# B&R Automation Studio project AsClientTest
Automation Studio 4.9

## Configuration Config1

CPU X20CP0484, AutomationRuntime H4.93, Build 4.1.2, Vc V4.72.6

### Task classes (Cpu.sw)
```
Cyclic#1 (cycle 5000 us, tolerance 10000000 us):
  uaCltTest <- uaCltTest.prg
Libraries: EasyUaClnt, AsIecCon, runtime, astime, AsOpcUac, standard, AsBrStr
```

### Hardware
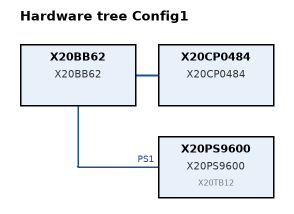
```
X20BB62 : X20BB62 v1.3.0.0
X20CP0484 : X20CP0484 v1.7.0.0  [SL -> X20BB62.SL1]
  Connector IF2:
    ActivateDevice = 1
    Mode = Manual
    InternetAddress = 192.168.2.10
    SubnetMask = 255.255.255.0
    ActivateSnmp = 2
  ConfigurationID = opcuaMethodCall_Config1
  Simulation = 1
  TimerDeviceType = SWIOTIMER
  TaskClassIdleTime = 10000
  CyclicTaskClassCount = 2
  Cyclic1Duration = 5000
  Cyclic1Tolerance = 10000000
  Cyclic2Duration = 20000
  Cyclic2Tolerance = 20000
  Cyclic3Duration = 50000
  Cyclic3Tolerance = 50000
  Cyclic4Duration = 100000
  Cyclic4Tolerance = 100000
  Cyclic5Duration = 200000
  Cyclic5Tolerance = 200000
  Cyclic6Duration = 500000
  Cyclic6Tolerance = 500000
  Cyclic7Duration = 1000000
  Cyclic7Tolerance = 1000000
  Cyclic8Duration = 10000
  Cyclic8Tolerance = 30000000
  FileDevice1
  FileDeviceName1 = USER
  FileDevicePath1 = USER_PATH
  ActivateOpcUa = 1
  OpcUaInformationModels_PV_Version = 1
X20PS9600 : X20PS9600 v1.6.1.0  [PS -> X20BB62.PS1; SS1 -> X20TB12.SS]
X20TB12 : X20TB12 v1.0.0.0
```

## Logical view

Binary libraries used (declarations not repeated): operator, runtime, astime, AsIecCon, EasyUaClnt 1.02.0, AsOpcUac, standard, AsBrStr


### Program Logical/uaCltTest (IEC)

#### Types.typ
```iecst
TYPE
	Sweep_typ : 	STRUCT
		input : Sweep_input_typ;
		output : Sweep_output_typ;
	END_STRUCT;
	Sweep_input_typ : 	STRUCT
		StartFrequency : LREAL;
		StopFrequency : LREAL;
		SweepPoints : DINT;
		SourceLevel : LREAL;
	END_STRUCT;
	Sweep_output_typ : 	STRUCT
		QFactor : LREAL;
		ResonanceFrequency : LREAL;
		Bandwidth : LREAL;
	END_STRUCT;
END_TYPE
```

#### Variables.var
```iecst
VAR CONSTANT
	MAX_OPCUA_CLIENTS : USINT := 9;
END_VAR
VAR
	EasyUaReads : ARRAY[0..MAX_OPCUA_CLIENTS] OF EasyUaRead;
	TON_0 : TON;
	Test : BOOL;
	i : USINT;
END_VAR
(*Variables to read into*)
VAR
	myBool : BOOL;
	myUsint : USINT;
	mySint : SINT;
	myUint : UINT;
	myInt : INT;
	myDint : DINT;
	myUdint : UDINT;
	myReal : REAL;
	myString : STRING[80];
END_VAR
```

#### Main.st
```iecst
// CLIENT SAMPLE TASK to read out the nodes from a OPCUA server.

PROGRAM _INIT
	// Setup for all clients
	FOR i:=0 TO MAX_OPCUA_CLIENTS DO
		EasyUaReads[i].ServerEndpointUrl := 'opc.tcp://127.0.0.2:4840'; // Don't use 127.0.0.1 as AS simulator put the server here as default.
		EasyUaReads[i].NamespaceUri := 'http://brdk.opcua.com';			// Specified on the server.
		EasyUaReads[i].NodeID.IdentifierType := UAIdentifierType_String;
	END_FOR

	// Setup for each node
	myBool;
	EasyUaReads[0].NodeID.Identifier := 'myBool';
	EasyUaReads[0].Variable := '::uaCltTest:myBool';

	myUsint;
	EasyUaReads[1].NodeID.Identifier := 'myUsint';
	EasyUaReads[1].Variable := '::uaCltTest:myUsint';

	mySint;
	EasyUaReads[2].NodeID.Identifier := 'mySint';
	EasyUaReads[2].Variable := '::uaCltTest:mySint';

	myUint;
	EasyUaReads[3].NodeID.Identifier := 'myUint';
	EasyUaReads[3].Variable := '::uaCltTest:myUint';

	myInt;
	EasyUaReads[4].NodeID.Identifier := 'myInt';
	EasyUaReads[4].Variable := '::uaCltTest:myInt';

	myDint;
	EasyUaReads[5].NodeID.Identifier := 'myDint';
	EasyUaReads[5].Variable := '::uaCltTest:myDint';

	myUdint;
	EasyUaReads[6].NodeID.Identifier := 'myUdint';
	EasyUaReads[6].Variable := '::uaCltTest:myUdint';

	myReal;
	EasyUaReads[7].NodeID.Identifier := 'myReal';
	EasyUaReads[7].Variable := '::uaCltTest:myReal';

	myString;
	EasyUaReads[8].NodeID.Identifier := 'myString';
	EasyUaReads[8].Variable := '::uaCltTest:myString';

	TON_0.PT := T#2s;

END_PROGRAM

PROGRAM _CYCLIC

	FOR i:=0 TO MAX_OPCUA_CLIENTS DO
		EasyUaReads[i]();
	END_FOR

END_PROGRAM

PROGRAM _EXIT
	FOR i:=0 TO MAX_OPCUA_CLIENTS DO
		EasyUaReads[i].Execute := FALSE;
		EasyUaReads[i]();
	END_FOR
END_PROGRAM
```

Listed in the project but not available here: Logical/Global.typ, Logical/Global.var
